{attribute 'GeneratedUsingTerminal: KL3361'}
{attribute addProperty BoxType "KL3361"}
{attribute addProperty Description ""}
{attribute addProperty Physics ""}
{attribute addProperty Id "Channel_1AT %Q*Channel_78571FB40"}
{attribute addProperty CRC "1942717114"}
{attribute addProperty Size "0"}
TYPE KL3361_73CB82BA :
STRUCT
	{attribute addProperty Name "Channel_1"}
	Channel_1 : Channel_78571FB4;
END_STRUCT
END_TYPE

(* stored: Version 1.2.0.0, ProductVersion 3.1.4024.9
   DUT KL3361_73CB82BA: Id {300a4be8-2887-4b61-adf9-b5f7d30d65e6} *)
